// TwinCAT 3 PLC project PLC
// ProgramVersion: 3.1.4026.1+972e9c44872ad038b353624a861fd7e3244e9f75
// libraries:
//   Tc2_Standard, * (Beckhoff Automation GmbH)
//   Tc2_System, * (Beckhoff Automation GmbH)
// project tree:
//   ChainOfResponsibility/ FB_Level1Handler.TcPOU, FB_Level2Handler.TcPOU, FB_Level3Handler.TcPOU, I_Handler.TcIO, PRG_SampleChainOfResponsibility.TcPOU
//   CommandPattern/interfaces/ I_Command.TcIO (not stored)
//   CommandPattern/receiver/ E_ColorCodes.TcDUT
//   CommandPattern/invoker/ FB_RemoteControl.TcPOU
//   CommandPattern/ PRG_SampleCommandPattern.TcPOU
//   CommandPattern/receiver/Light/commands/ FB_CmdLightChangeBrightness.TcPOU, FB_CmdLightChangeColor.TcPOU, FB_CmdLightOff.TcPOU, FB_CmdLightOn.TcPOU
//   CommandPattern/receiver/Light/ FB_Light.TcPOU, I_Light.TcIO
//   Iterator/Collections/ FB_ElementsStation1.TcPOU, FB_ElementsStation2.TcPOU
//   Iterator/Element/ FB_ElementIterator.TcPOU, I_ElementIterator.TcIO, I_IterableElementCollection.TcIO, ST_Element.TcDUT
//   Iterator/ PRG_SampleIterator.TcPOU
//   / MAIN.TcPOU, PlcTask.TcTTO
//   Mediator/Components/Heater/ FB_Heater.TcPOU, I_Heater.TcIO
//   Mediator/Components/SimulateRoomTemperature/ FB_SimulateTemperature.TcPOU
//   Mediator/Components/Thermostat/ FB_Thermostat.TcPOU, I_Thermostat.TcIO
//   Mediator/Mediator/ FB_SmartHome.TcPOU, I_Mediator.TcIO
//   Mediator/ PRG_SampleMediator.TcPOU
//   Memento/Caretaker/ FB_DocumentCaretaker.TcPOU
//   Memento/Memento/ ST_DocumentMemento.TcDUT
//   Memento/Originator/ FB_Document.TcPOU
//   Memento/ PRG_SampleMemento.TcPOU
//   Observer/ PRG_SampleObserver.TcPOU
//   Observer/Publisher/ FB_Publisher.TcPOU
//   Observer/Subscriber/ FB_Subscriber.TcPOU, I_Subscriber.TcIO
//   StatePattern/ FB_StateMachine.TcPOU, PRG_SampleState.TcPOU
//   StatePattern/States/ FB_NotReadyState.TcPOU, FB_ProcessingState.TcPOU, FB_ReadyState.TcPOU, I_State.TcIO
//   Strategy/ FB_TravelTimeCalculator.TcPOU, PRG_SampleStrategy.TcPOU
//   Strategy/Strategies/ FB_StrategyTravelByTrain.TcPOU, FB_StrategyTravelByCar.TcPOU, FB_StrategyTravelByBycicle.TcPOU, I_Strategy.TcIO
//   Visitor/ FB_ElementA.TcPOU, FB_ElementB.TcPOU, FB_Visitor.TcPOU, I_VisitibleElement.TcIO, I_Visitor.TcIO, PRG_SampleVisitor.TcPOU
// real-time tasks:
//   TASK PlcTask: cycle T#10ms, priority 20, ADS port 350

CONFIGURATION PLC
    RESOURCE PLC ON TwinCAT3
        TASK PlcTask(INTERVAL := T#10ms, PRIORITY := 20);
        PROGRAM MAIN WITH PlcTask : MAIN;
    END_RESOURCE
END_CONFIGURATION

// ---- CommandPattern/receiver/E_ColorCodes.TcDUT
{attribute 'qualified_only'}
{attribute 'to_string'}
TYPE E_ColorCodes :
(
	Black 	:= 16#000000,
	Red		:= 16#FF0000,
	Maroon	:= 16#800000,
	Yellow	:= 16#FFFF00,
	Olive	:= 16#808000,
	Lime	:= 16#00FF00,
	Green	:= 16#008000,
	Aqua	:= 16#00FFFF,
	Teal	:= 16#008080,
	Blue	:= 16#0000FF,
	Navy	:= 16#000080,	
	Fuchsia	:= 16#FF00FF,	
	Purple	:= 16#800080,
	White	:= 16#FFFFFF,
	Silver	:= 16#C0C0C0,
	Gray	:= 16#808080
)DWORD;
END_TYPE

// ---- Iterator/Element/ST_Element.TcDUT
TYPE ST_Element :
STRUCT
	sName		:STRING;
END_STRUCT
END_TYPE

// ---- Memento/Memento/ST_DocumentMemento.TcDUT
TYPE ST_DocumentMemento :
STRUCT
	sContent		: STRING;
END_STRUCT
END_TYPE

// ---- ChainOfResponsibility/I_Handler.TcIO
INTERFACE I_Handler

METHOD handleRequest : BOOL
VAR_INPUT
	in_sRequest		: STRING;
END_VAR
END_METHOD

END_INTERFACE

// ---- CommandPattern/receiver/Light/I_Light.TcIO
INTERFACE I_Light

PROPERTY bIsOn : BOOL
GET
END_GET
END_PROPERTY

METHOD changeBrightness : BOOL
VAR_INPUT
	in_rNewBrightness	:REAL;
END_VAR
END_METHOD

METHOD changeColor : BOOL
VAR_INPUT
	in_eNewColor	:E_ColorCodes;
END_VAR
END_METHOD

PROPERTY eColor : E_ColorCodes
GET
END_GET
END_PROPERTY

PROPERTY rBrightness : REAL
GET
END_GET
END_PROPERTY

METHOD turnLightOff : BOOL
VAR_INPUT
END_VAR
END_METHOD

METHOD turnLightOn : BOOL
VAR_INPUT
END_VAR
END_METHOD

END_INTERFACE

// ---- Iterator/Element/I_ElementIterator.TcIO
INTERFACE I_ElementIterator

METHOD hasNext : BOOL
VAR_INPUT
END_VAR
END_METHOD

METHOD init : BOOL
VAR_IN_OUT
	io_astElements	:ARRAY[*] OF ST_Element;
END_VAR
END_METHOD

METHOD next : ST_Element;
VAR_INPUT
END_VAR
END_METHOD

END_INTERFACE

// ---- Iterator/Element/I_IterableElementCollection.TcIO
INTERFACE I_IterableElementCollection

METHOD createIterator : REFERENCE TO FB_ElementIterator
VAR_INPUT
END_VAR
END_METHOD

END_INTERFACE

// ---- Mediator/Components/Heater/I_Heater.TcIO
INTERFACE I_Heater

PROPERTY bIsOn : BOOL
GET
END_GET
END_PROPERTY

PROPERTY sLocation : STRING
GET
END_GET
END_PROPERTY

PROPERTY sName : String
GET
END_GET
END_PROPERTY

METHOD turnOff : Bool
VAR_INPUT
END_VAR
END_METHOD

METHOD turnOn : Bool
VAR_INPUT
END_VAR
END_METHOD

END_INTERFACE

// ---- Mediator/Components/Thermostat/I_Thermostat.TcIO
INTERFACE I_Thermostat

PROPERTY rRequestedTemperature : REAL
GET
END_GET
SET
END_SET
END_PROPERTY

PROPERTY rTemperature : REAL
GET
END_GET
END_PROPERTY

PROPERTY sLocation : STRING
GET
END_GET
END_PROPERTY

PROPERTY sName : String
GET
END_GET
END_PROPERTY

END_INTERFACE

// ---- Mediator/Mediator/I_Mediator.TcIO
INTERFACE I_Mediator

METHOD notify : BOOL
VAR_INPUT
	in_sSenderName		: STRING;
	in_sEvent 			: STRING;
END_VAR
END_METHOD

END_INTERFACE

// ---- Observer/Subscriber/I_Subscriber.TcIO
INTERFACE I_Subscriber

METHOD update : BOOL
VAR_INPUT
	in_sContent			: STRING;
END_VAR
END_METHOD

END_INTERFACE

// ---- StatePattern/States/I_State.TcIO
INTERFACE I_State

PROPERTY CurrentState : STRING
GET
END_GET
END_PROPERTY

METHOD ErrorGone
VAR_INPUT
END_VAR
END_METHOD

METHOD ErrorOccured
VAR_INPUT
END_VAR
END_METHOD

METHOD StartProcess
VAR_INPUT
END_VAR
END_METHOD

METHOD StopProcess
VAR_INPUT
END_VAR
END_METHOD

END_INTERFACE

// ---- Strategy/Strategies/I_Strategy.TcIO
INTERFACE I_Strategy

METHOD execute
VAR_INPUT
	in_rDistance		:REAL;
END_VAR
END_METHOD

END_INTERFACE

// ---- Visitor/I_VisitibleElement.TcIO
INTERFACE I_VisitibleElement

METHOD accept
VAR_INPUT
	in_ipVisitor	: I_Visitor;
END_VAR
END_METHOD

END_INTERFACE

// ---- Visitor/I_Visitor.TcIO
INTERFACE I_Visitor

METHOD VisitElementA
VAR_INPUT
	in_fbElementA		:FB_ElementA;
END_VAR
END_METHOD

METHOD VisitElementB
VAR_INPUT
	in_fbElementB		:FB_ElementB;
END_VAR
END_METHOD

END_INTERFACE

// ---- MAIN.TcPOU
PROGRAM MAIN
VAR
END_VAR

//*************************************************************
// Chain of Responsibility
//*************************************************************
	PRG_SampleChainOfResponsibility();

//*************************************************************
// Command Pattern 
//*************************************************************
	PRG_SampleCommandPattern();
	
//*************************************************************
// Iterator Pattern 
//*************************************************************
	PRG_SampleIterator();

//*************************************************************
// Mediator Pattern 
//*************************************************************
	PRG_SampleMediator();
	
//*************************************************************
// Memento Pattern 
//*************************************************************
	PRG_SampleMemento();
	
//*************************************************************
// Observer Pattern 
//*************************************************************
	PRG_SampleObserver();
	
//*************************************************************
// State Pattern 
//*************************************************************
	PRG_SampleState();	
	
//*************************************************************
// Strategy Pattern 
//*************************************************************
	PRG_SampleStrategy();

END_PROGRAM

// ---- ChainOfResponsibility/PRG_SampleChainOfResponsibility.TcPOU
PROGRAM PRG_SampleChainOfResponsibility
VAR
	fbLvl1Handler			: FB_Level1Handler();
	fbLvl2Handler			: FB_Level2Handler();
	fbLvl3Handler			: FB_Level3Handler();
	
	
	sRequest				: STRING;
	sOldRequest				: STRING;
	bRequestHandled			: BOOL;
	aipHandlers				: ARRAY[0..2] OF I_Handler;
	iCurrentHandlerIndex	: INT;
END_VAR

//*************************************************************
// Call initial Request
//*************************************************************
IF sRequest <> sOldRequest THEN
	sOldRequest := sRequest;
	
	aipHandlers[0] := fbLvl1Handler;
	aipHandlers[1] := fbLvl2Handler;
	aipHandlers[2] := fbLvl3Handler;
	bRequestHandled := FALSE;
	
	FOR iCurrentHandlerIndex:= 0 TO 2 DO
		bRequestHandled := aipHandlers[iCurrentHandlerIndex].handleRequest(in_sRequest := sRequest);
		IF bRequestHandled THEN
			EXIT;
		END_IF
	END_FOR
	
	IF NOT bRequestHandled THEN
		ADSLOGSTR(msgCtrlMask:= ADSLOG_MSGTYPE_ERROR, msgFmtStr:= 'Request cannot be solved by anyone. Request: %s', strArg:= sRequest);
	END_IF
END_IF

END_PROGRAM

// ---- ChainOfResponsibility/FB_Level1Handler.TcPOU
FUNCTION_BLOCK FB_Level1Handler IMPLEMENTS I_Handler
VAR_INPUT
END_VAR
VAR_OUTPUT
END_VAR
VAR
END_VAR

METHOD handleRequest : BOOL
VAR_INPUT
	in_sRequest		: STRING;
END_VAR
handleRequest := FALSE;

IF FIND(in_sRequest, 'Level 1') <> 0 THEN
	ADSLOGSTR(msgCtrlMask:= ADSLOG_MSGTYPE_ERROR, msgFmtStr:= 'Request solved by Level 1. Request: %s', strArg:= in_sRequest);
	handleRequest := TRUE;
ELSE
	ADSLOGSTR(msgCtrlMask:= ADSLOG_MSGTYPE_ERROR, msgFmtStr:= 'Request cannot solved by Level 1. Request: %s', strArg:= in_sRequest);
END_IF
END_METHOD

END_FUNCTION_BLOCK

// ---- ChainOfResponsibility/FB_Level2Handler.TcPOU
FUNCTION_BLOCK FB_Level2Handler IMPLEMENTS I_Handler
VAR_INPUT
END_VAR
VAR_OUTPUT
END_VAR
VAR
END_VAR

METHOD handleRequest : BOOL
VAR_INPUT
	in_sRequest		: STRING;
END_VAR
handleRequest := FALSE;

IF FIND(in_sRequest, 'Level 2') <> 0 THEN
	ADSLOGSTR(msgCtrlMask:= ADSLOG_MSGTYPE_ERROR, msgFmtStr:= 'Request solved by Level 2. Request: %s', strArg:= in_sRequest);
	handleRequest := TRUE;
ELSE
	ADSLOGSTR(msgCtrlMask:= ADSLOG_MSGTYPE_ERROR, msgFmtStr:= 'Request cannot be solved by Level 2. Request: %s', strArg:= in_sRequest);
END_IF
END_METHOD

END_FUNCTION_BLOCK

// ---- ChainOfResponsibility/FB_Level3Handler.TcPOU
FUNCTION_BLOCK FB_Level3Handler IMPLEMENTS I_Handler
VAR_INPUT
END_VAR
VAR_OUTPUT
END_VAR
VAR
END_VAR

METHOD handleRequest : BOOL
VAR_INPUT
	in_sRequest		: STRING;
END_VAR
handleRequest := FALSE;

IF FIND(in_sRequest, 'Level 3') <> 0 THEN
	ADSLOGSTR(msgCtrlMask:= ADSLOG_MSGTYPE_ERROR, msgFmtStr:= 'Request solved by Level 3. Request: %s', strArg:= in_sRequest);
	handleRequest := TRUE;
ELSE
	ADSLOGSTR(msgCtrlMask:= ADSLOG_MSGTYPE_ERROR, msgFmtStr:= 'Request cannot solved by Level 3. Request: %s', strArg:= in_sRequest);
END_IF
END_METHOD

END_FUNCTION_BLOCK

// ---- CommandPattern/PRG_SampleCommandPattern.TcPOU
PROGRAM PRG_SampleCommandPattern
VAR
	fbLight								: FB_Light;
	// Commands
	fbLightOnCmd						: FB_CmdLightOn(ipLight := fbLight);
	fbLightOffCmd						: FB_CmdLightOff(ipLight := fbLight);
	fbIncreaseBrightnessCmd				: FB_CmdLightChangeBrightness(ipLight := fbLight, rBrightnessChange:= 10.0);
	fbDecreaseBrightnessCmd				: FB_CmdLightChangeBrightness(ipLight := fbLight, rBrightnessChange:= -10.0);
	fbChangeColorFav1Cmd				: FB_CmdLightChangeColor(ipLight := fbLight, eColor:= E_ColorCodes.Red);
	fbChangeColorFav2Cmd				: FB_CmdLightChangeColor(ipLight := fbLight, eColor:= E_ColorCodes.Green);
	// Invoker
	fbRemoteControl						: FB_RemoteControl(ipCmdOn:= fbLightOnCmd, ipCmdOff:= fbLightOffCmd, ipCmdFav1:= fbIncreaseBrightnessCmd, ipCmdFav2:= fbDecreaseBrightnessCmd);
	
	// Test events
	bChangeToColorControl				: BOOL;
	bChangeToBrightnessControl			: BOOL;
	
	eOldFav1Color						: E_ColorCodes;
	eFav1Color							: E_ColorCodes;	
	eOldFav2Color						: E_ColorCodes;
	eFav2Color							: E_ColorCodes;
	
	rOldIncreaseSteps					: REAL;
	rIncreaseSteps						: REAL;	
	rOldDecreaseSteps					: REAL;
	rDecreaseSteps						: REAL;	
	
	bPressOn							: BOOL;
	bPressOff							: BOOL;
	bPressFav1							: BOOL;
	bPressFav2							: BOOL;
END_VAR

//*************************************************************
// Call Object Light
//*************************************************************
	fbLight();

//*************************************************************
// Change Functionality of Remote Control
//*************************************************************

	//*************************************************************
	// Color control
	//*************************************************************
	IF bChangeToColorControl THEN
		bChangeToColorControl := FALSE;
		fbRemoteControl.setCommands(
										in_ipCmdOn		:= fbLightOnCmd, 
										in_ipCmdOff		:= fbLightOffCmd, 
										in_ipCmdFav1	:= fbChangeColorFav1Cmd, 
										in_ipCmdFav2	:= fbChangeColorFav2Cmd);
	END_IF
	
	IF eFav1Color <> eOldFav1Color THEN
		eOldFav1Color := eFav1Color;
		fbChangeColorFav1Cmd.setChangeColor(in_eNewChangeColor := eFav1Color);
	END_IF
	
	IF eFav2Color <> eOldFav2Color THEN
		eOldFav2Color := eFav2Color;
		fbChangeColorFav2Cmd.setChangeColor(in_eNewChangeColor := eFav2Color);
	END_IF
	
	//*************************************************************
	// Brightness control
	//*************************************************************
	IF bChangeToBrightnessControl THEN
		bChangeToBrightnessControl := FALSE;
		fbRemoteControl.setCommands(
										in_ipCmdOn		:= fbLightOnCmd, 
										in_ipCmdOff		:= fbLightOffCmd, 
										in_ipCmdFav1	:= fbIncreaseBrightnessCmd, 
										in_ipCmdFav2	:= fbDecreaseBrightnessCmd);
	END_IF
	
	IF rIncreaseSteps <> rOldIncreaseSteps THEN
		rOldIncreaseSteps := rIncreaseSteps;
		fbIncreaseBrightnessCmd.setChangeBrightness(in_rNewChangeBrightness := rIncreaseSteps);
	END_IF
	
	IF rDecreaseSteps <> rOldDecreaseSteps THEN
		rOldDecreaseSteps := rDecreaseSteps;
		fbDecreaseBrightnessCmd.setChangeBrightness(in_rNewChangeBrightness := rDecreaseSteps);
	END_IF

//*************************************************************
// Do Actions
//*************************************************************
	IF bPressOn THEN
		bPressOn := FALSE;
		fbRemoteControl.pressOn();
	END_IF
	
	IF bPressOff THEN
		bPressOff := FALSE;
		fbRemoteControl.pressOff();
	END_IF
	
	IF bPressFav1 THEN
		bPressFav1 := FALSE;
		fbRemoteControl.pressFav1();
	END_IF
	
	IF bPressFav2 THEN
		bPressFav2 := FALSE;
		fbRemoteControl.pressFav2();
	END_IF

END_PROGRAM

// ---- CommandPattern/receiver/Light/FB_Light.TcPOU
FUNCTION_BLOCK FB_Light IMPLEMENTS I_LIGHT
VAR_INPUT
END_VAR
VAR_OUTPUT
END_VAR
VAR
	_rBrightness	: REAL;
	_eColor			: E_ColorCodes;
	_bIsOn			: BOOL;
END_VAR

PROPERTY bIsOn : BOOL
GET
bIsOn := _bIsOn;
END_GET
END_PROPERTY

METHOD changeBrightness : BOOL
VAR_INPUT
	in_rNewBrightness	: REAL;
END_VAR
IF in_rNewBrightness > 100.0 THEN
	_rBrightness := 100.0;
ELSIF in_rNewBrightness < 0.0 THEN
	_rBrightness := 0.0;
ELSE
	_rBrightness := in_rNewBrightness;
END_IF

ADSLOGSTR(msgCtrlMask:= ADSLOG_MSGTYPE_ERROR, msgFmtStr:= 'New Brightness: %s', strArg:= TO_STRING(_rBrightness));
END_METHOD

METHOD changeColor : BOOL
VAR_INPUT
	in_eNewColor	:E_ColorCodes;
END_VAR
_eColor := in_eNewColor;
ADSLOGSTR(msgCtrlMask:= ADSLOG_MSGTYPE_ERROR, msgFmtStr:= 'New Color: %s', strArg:= TO_STRING(_eColor));
END_METHOD

PROPERTY eColor : E_ColorCodes
GET
eColor := _eColor;
END_GET
END_PROPERTY

PROPERTY rBrightness : REAL
GET
rBrightness := _rBrightness;
END_GET
END_PROPERTY

METHOD turnLightOff : BOOL
VAR_INPUT
END_VAR
_bIsOn := FALSE;
ADSLOGSTR(msgCtrlMask:= ADSLOG_MSGTYPE_ERROR, msgFmtStr:= 'Light is off', strArg:= '');
ADSLOGSTR(msgCtrlMask:= ADSLOG_MSGTYPE_ERROR, msgFmtStr:= 'Brightness: %s', strArg:= TO_STRING(_rBrightness));
ADSLOGSTR(msgCtrlMask:= ADSLOG_MSGTYPE_ERROR, msgFmtStr:= 'Color: %s', strArg:= TO_STRING(_eColor));
END_METHOD

METHOD turnLightOn : BOOL
VAR_INPUT
END_VAR
_bIsOn := TRUE;

IF _rBrightness <= 0.0 THEN
	_rBrightness := 100.0;
END_IF

IF _eColor = E_ColorCodes.Black THEN
	_eColor := E_ColorCodes.White;
END_IF

ADSLOGSTR(msgCtrlMask:= ADSLOG_MSGTYPE_ERROR, msgFmtStr:= 'Light is on', strArg:= '');
ADSLOGSTR(msgCtrlMask:= ADSLOG_MSGTYPE_ERROR, msgFmtStr:= 'Brightness: %s', strArg:= TO_STRING(_rBrightness));
ADSLOGSTR(msgCtrlMask:= ADSLOG_MSGTYPE_ERROR, msgFmtStr:= 'Color: %s', strArg:= TO_STRING(_eColor));
END_METHOD

END_FUNCTION_BLOCK

// ---- CommandPattern/receiver/Light/commands/FB_CmdLightOn.TcPOU
FUNCTION_BLOCK FB_CmdLightOn IMPLEMENTS I_Command
VAR_INPUT
END_VAR
VAR_OUTPUT
END_VAR
VAR
	_ipLight				: I_Light;
END_VAR

METHOD execute : BOOL
_ipLight.turnLightOn();
END_METHOD

//FB_Init is always available implicitly and it is used primarily for initialization.
//The return value is not evaluated. For a specific influence, you can also declare the
//methods explicitly and provide additional code there with the standard initialization
//code. You can evaluate the return value.
METHOD FB_Init: BOOL
VAR_INPUT
    bInitRetains: BOOL; // TRUE: the retain variables are initialized (reset warm / reset cold)
    bInCopyCode: BOOL;  // TRUE: the instance will be copied to the copy code afterward (online change)   
	ipLight: I_Light;
END_VAR
_ipLight := ipLight;
END_METHOD

END_FUNCTION_BLOCK

// ---- CommandPattern/receiver/Light/commands/FB_CmdLightOff.TcPOU
FUNCTION_BLOCK FB_CmdLightOff IMPLEMENTS I_Command
VAR_INPUT
END_VAR
VAR_OUTPUT
END_VAR
VAR
	_ipLight				: I_Light;
END_VAR

METHOD execute : BOOL
_ipLight.turnLightOff();
END_METHOD

//FB_Init is always available implicitly and it is used primarily for initialization.
//The return value is not evaluated. For a specific influence, you can also declare the
//methods explicitly and provide additional code there with the standard initialization
//code. You can evaluate the return value.
METHOD FB_Init: BOOL
VAR_INPUT
    bInitRetains: BOOL; // TRUE: the retain variables are initialized (reset warm / reset cold)
    bInCopyCode: BOOL;  // TRUE: the instance will be copied to the copy code afterward (online change)   
	ipLight: I_Light;
END_VAR
_ipLight := ipLight;
END_METHOD

END_FUNCTION_BLOCK

// ---- CommandPattern/receiver/Light/commands/FB_CmdLightChangeBrightness.TcPOU
FUNCTION_BLOCK FB_CmdLightChangeBrightness IMPLEMENTS I_Command
VAR_INPUT
END_VAR
VAR_OUTPUT
END_VAR
VAR
	_rBrightnessChange		: REAL;
	_ipLight				: I_Light;
END_VAR

METHOD execute : BOOL
_ipLight.changeBrightness(in_rNewBrightness:= (_ipLight.rBrightness + _rBrightnessChange));
END_METHOD

//FB_Init is always available implicitly and it is used primarily for initialization.
//The return value is not evaluated. For a specific influence, you can also declare the
//methods explicitly and provide additional code there with the standard initialization
//code. You can evaluate the return value.
METHOD FB_Init: BOOL
VAR_INPUT
    bInitRetains: BOOL; // TRUE: the retain variables are initialized (reset warm / reset cold)
    bInCopyCode: BOOL;  // TRUE: the instance will be copied to the copy code afterward (online change)   
	rBrightnessChange :REAL;
	ipLight: I_Light;
END_VAR
_ipLight := ipLight;
_rBrightnessChange := rBrightnessChange;
END_METHOD

METHOD setChangeBrightness : BOOL
VAR_INPUT
	in_rNewChangeBrightness	: REAL;
END_VAR
_rBrightnessChange := in_rNewChangeBrightness;
END_METHOD

END_FUNCTION_BLOCK

// ---- CommandPattern/receiver/Light/commands/FB_CmdLightChangeColor.TcPOU
FUNCTION_BLOCK FB_CmdLightChangeColor IMPLEMENTS I_Command
VAR_INPUT
END_VAR
VAR_OUTPUT
END_VAR
VAR
	_eChangeColor			: E_ColorCodes;
	_ipLight				: I_Light;
END_VAR

METHOD execute : BOOL
_ipLight.changeColor(in_eNewColor:= _eChangeColor);
END_METHOD

//FB_Init is always available implicitly and it is used primarily for initialization.
//The return value is not evaluated. For a specific influence, you can also declare the
//methods explicitly and provide additional code there with the standard initialization
//code. You can evaluate the return value.
METHOD FB_Init: BOOL
VAR_INPUT
    bInitRetains: BOOL; // TRUE: the retain variables are initialized (reset warm / reset cold)
    bInCopyCode: BOOL;  // TRUE: the instance will be copied to the copy code afterward (online change)   
	eColor : E_ColorCodes;
	ipLight: I_Light;
END_VAR
_ipLight := ipLight;
_eChangeColor := eColor;
END_METHOD

METHOD setChangeColor : BOOL
VAR_INPUT
	in_eNewChangeColor	: E_ColorCodes;
END_VAR
_eChangeColor := in_eNewChangeColor;
END_METHOD

END_FUNCTION_BLOCK

// ---- CommandPattern/invoker/FB_RemoteControl.TcPOU
FUNCTION_BLOCK FB_RemoteControl
VAR_INPUT
END_VAR
VAR_OUTPUT
END_VAR
VAR
	_ipCmdOn		: I_Command;
	_ipCmdOff		: I_Command;
	_ipCmdFav1		: I_Command;
	_ipCmdFav2		: I_Command;
END_VAR

//FB_Init is always available implicitly and it is used primarily for initialization.
//The return value is not evaluated. For a specific influence, you can also declare the
//methods explicitly and provide additional code there with the standard initialization
//code. You can evaluate the return value.
METHOD FB_Init: BOOL
VAR_INPUT
    bInitRetains: BOOL; // TRUE: the retain variables are initialized (reset warm / reset cold)
    bInCopyCode: BOOL;  // TRUE: the instance will be copied to the copy code afterward (online change)   
	ipCmdOn		: I_Command;
	ipCmdOff	: I_Command;
	ipCmdFav1	: I_Command;
	ipCmdFav2	: I_Command;
END_VAR
_ipCmdOn		:= ipCmdOn;
_ipCmdOff		:= ipCmdOff;
_ipCmdFav1		:= ipCmdFav1;
_ipCmdFav2		:= ipCmdFav2;
END_METHOD

METHOD pressFav1 : BOOL
VAR_INPUT
END_VAR
_ipCmdFav1.execute();
END_METHOD

METHOD pressFav2 : BOOL
VAR_INPUT
END_VAR
_ipCmdFav2.execute();
END_METHOD

METHOD pressOff : BOOL
VAR_INPUT
END_VAR
_ipCmdOff.execute();
END_METHOD

METHOD pressOn : BOOL
VAR_INPUT
END_VAR
_ipCmdOn.execute();
END_METHOD

METHOD setCommands : BOOL
VAR_INPUT
	in_ipCmdOn		: I_Command;
	in_ipCmdOff		: I_Command;
	in_ipCmdFav1	: I_Command;
	in_ipCmdFav2	: I_Command;
END_VAR
_ipCmdOn		:= in_ipCmdOn;
_ipCmdOff		:= in_ipCmdOff;
_ipCmdFav1		:= in_ipCmdFav1;
_ipCmdFav2		:= in_ipCmdFav2;
END_METHOD

END_FUNCTION_BLOCK

// ---- Iterator/PRG_SampleIterator.TcPOU
PROGRAM PRG_SampleIterator
VAR
	fbElementsStation1				: FB_ElementsStation1;
	fbElementStation1Iterator   	: REFERENCE TO FB_ElementIterator;
	fbElementsStation2				: FB_ElementsStation2;
	fbElementStation2Iterator   	: REFERENCE TO FB_ElementIterator;
	
	bIterateStation1				: BOOL;
	bIterateStation2				: BOOL;
END_VAR

VAR_TEMP
	stElement						:ST_Element;
END_VAR

fbElementsStation1();
fbElementsStation2();


IF bIterateStation1 THEN
	bIterateStation1 := FALSE;
	
	fbElementStation1Iterator REF= fbElementsStation1.createIterator();
	WHILE fbElementStation1Iterator.hasNext() DO
		stElement := fbElementStation1Iterator.next();
		ADSLOGSTR(msgCtrlMask:= ADSLOG_MSGTYPE_ERROR, msgFmtStr:= '%s found.', strArg:= stElement.sName);
	END_WHILE
END_IF

IF bIterateStation2 THEN
	bIterateStation2 := FALSE;
	
	fbElementStation2Iterator REF= fbElementsStation2.createIterator();
	WHILE fbElementStation2Iterator.hasNext() DO
		stElement := fbElementStation2Iterator.next();
		ADSLOGSTR(msgCtrlMask:= ADSLOG_MSGTYPE_ERROR, msgFmtStr:= '%s found.', strArg:= stElement.sName);
	END_WHILE
END_IF

END_PROGRAM

// ---- Iterator/Collections/FB_ElementsStation1.TcPOU
FUNCTION_BLOCK FB_ElementsStation1 IMPLEMENTS I_IterableElementCollection
VAR_INPUT
END_VAR
VAR_OUTPUT
END_VAR
VAR
	_astElements			: ARRAY[0..MAX_ELEMENTS] OF ST_Element;	
	_fbIterator				: FB_ElementIterator;
END_VAR

VAR CONSTANT
	MAX_ELEMENTS			: INT := 30;
END_VAR

METHOD createIterator : REFERENCE TO FB_ElementIterator
_fbIterator.init(io_astElements := _astElements);
createIterator REF= _fbIterator;
END_METHOD

//FB_Init is always available implicitly and it is used primarily for initialization.
//The return value is not evaluated. For a specific influence, you can also declare the
//methods explicitly and provide additional code there with the standard initialization
//code. You can evaluate the return value.
METHOD FB_Init: BOOL
VAR_INPUT
    bInitRetains: BOOL; // TRUE: the retain variables are initialized (reset warm / reset cold)
    bInCopyCode: BOOL;  // TRUE: the instance will be copied to the copy code afterward (online change)   
END_VAR
VAR 
	i : INT;
END_VAR
FOR i:= 0 TO MAX_ELEMENTS DO
	_astElements[i].sName:= CONCAT('Element Station 1 No: ', TO_STRING(i + 1));
END_FOR
END_METHOD

END_FUNCTION_BLOCK

// ---- Iterator/Element/FB_ElementIterator.TcPOU
FUNCTION_BLOCK FB_ElementIterator IMPLEMENTS I_ElementIterator
VAR_INPUT
END_VAR
VAR_OUTPUT
END_VAR
VAR
	_pElementData		: POINTER TO ST_Element;
	_diNumOfElements	: DINT;
	_diIndex			: DINT;
END_VAR

METHOD hasNext : BOOL
VAR
	
END_VAR
IF _pElementData = 0 THEN
	RETURN;
END_IF

hasNext := _diIndex < _diNumOfElements;
END_METHOD

METHOD init : BOOL
VAR_IN_OUT
	io_astElements	:ARRAY[*] OF ST_Element;
END_VAR
_pElementData 		:= io_astElements;
_diNumOfElements 	:= UPPER_BOUND(io_astElements, 1);
_diIndex			:= LOWER_BOUND(io_astElements, 1);
END_METHOD

METHOD next : ST_Element
VAR
	stElement :ST_Element;
END_VAR
IF _pElementData = 0 THEN
	RETURN;
END_IF

IF _diIndex < _diNumOfElements THEN
	MEMCPY(srcAddr:= (_pElementData + (_diIndex * SIZEOF(stElement))), destAddr:= ADR(stElement), n:= SIZEOF(stElement));
	next := stElement;
	_diIndex := _diIndex + 1;
END_IF
END_METHOD

END_FUNCTION_BLOCK

// ---- Iterator/Collections/FB_ElementsStation2.TcPOU
FUNCTION_BLOCK FB_ElementsStation2 IMPLEMENTS I_IterableElementCollection
VAR_INPUT
END_VAR
VAR_OUTPUT
END_VAR
VAR
	_astElements			: ARRAY[0..MAX_ELEMENTS] OF ST_Element;
	_fbIterator				: FB_ElementIterator;
END_VAR

VAR CONSTANT
	MAX_ELEMENTS			: INT := 5;
END_VAR

METHOD createIterator : REFERENCE TO FB_ElementIterator
_fbIterator.init(io_astElements := _astElements);
createIterator REF= _fbIterator;
END_METHOD

//FB_Init is always available implicitly and it is used primarily for initialization.
//The return value is not evaluated. For a specific influence, you can also declare the
//methods explicitly and provide additional code there with the standard initialization
//code. You can evaluate the return value.
METHOD FB_Init: BOOL
VAR_INPUT
    bInitRetains: BOOL; // TRUE: the retain variables are initialized (reset warm / reset cold)
    bInCopyCode: BOOL;  // TRUE: the instance will be copied to the copy code afterward (online change)   
END_VAR
VAR 
	i : INT;
END_VAR
FOR i:= 0 TO MAX_ELEMENTS DO
	_astElements[i].sName:= CONCAT('Element Station 2 No: ', TO_STRING(i + 1));
END_FOR
END_METHOD

END_FUNCTION_BLOCK

// ---- Mediator/PRG_SampleMediator.TcPOU
PROGRAM PRG_SampleMediator
VAR
	fbSmartHomeDevice			:FB_SmartHome;	

	fbHeaterKitchen				:FB_Heater(sName:= 'Heater', sLocation := 'Kitchen', ipMediator:= fbSmartHomeDevice);
	fbHeaterBedroom				:FB_Heater(sName:= 'Heater', sLocation := 'Bedroom', ipMediator:= fbSmartHomeDevice);
	
	fbThermostatKitchen			:FB_Thermostat(sName:= 'Thermostat', sLocation := 'Kitchen', rRequestedTemperature := 20.0, ipMediator:= fbSmartHomeDevice);
	fbThermostatBedroom			:FB_Thermostat(sName:= 'Door', sLocation := 'Bedroom', rRequestedTemperature := 14.0, ipMediator:= fbSmartHomeDevice);
	
	fbRoomTempKitchen			:FB_SimulateTemperature;
	fbRoomTempBedroom			:FB_SimulateTemperature;
	
	bEnable						:BOOL;
	bAddAllDevices				:BOOL := TRUE; // Event to add all devices to Mediator
	bRemoveAllDevices			:BOOL;
END_VAR

//*************************************************************
// Disable Test enviroment
//*************************************************************	
	IF NOT bEnable THEN
		
		RETURN;
		
	END_IF

//*************************************************************
// Call Objects
//*************************************************************
	fbSmartHomeDevice();
	
	fbHeaterKitchen();
	fbHeaterBedroom();
	
	fbThermostatKitchen(in_rTemperature := fbRoomTempKitchen.out_bSimTemperature);
	fbThermostatBedroom(in_rTemperature := fbRoomTempBedroom.out_bSimTemperature);
	
	fbRoomTempKitchen(in_bTempShouldRise := fbHeaterKitchen.bIsOn);
	fbRoomTempBedroom(in_bTempShouldRise := fbHeaterBedroom.bIsOn);
	
//*************************************************************
// Add Objects to Smart Home Device
//*************************************************************	
IF bAddAllDevices THEN
	
	bAddAllDevices := FALSE;
	
	fbSmartHomeDevice.addHeater(fbHeaterKitchen);
	//fbSmartHomeDevice.addHeater(fbHeaterBedroom);
	
	fbSmartHomeDevice.addThermostat(fbThermostatKitchen);
	//fbSmartHomeDevice.addThermostat(fbThermostatBedroom);
	
END_IF

IF bRemoveAllDevices THEN
	
	bRemoveAllDevices := FALSE;
	
	fbSmartHomeDevice.removeHeater(fbHeaterKitchen);
	fbSmartHomeDevice.removeHeater(fbHeaterBedroom);
	
	fbSmartHomeDevice.removeThermostat(fbThermostatKitchen);
	fbSmartHomeDevice.removeThermostat(fbThermostatBedroom);
	
END_IF

END_PROGRAM

// ---- Mediator/Mediator/FB_SmartHome.TcPOU
FUNCTION_BLOCK FB_SmartHome IMPLEMENTS I_Mediator
VAR_INPUT
END_VAR
VAR_OUTPUT
END_VAR
VAR
	_aipHeater				: ARRAY [0..MAX_HEATER] OF I_Heater;
	_aipThermostat			: ARRAY [0..MAX_THERMOSTAT] OF I_Thermostat;
END_VAR
VAR CONSTANT
	MAX_HEATER				: INT := 5;
	MAX_THERMOSTAT			: INT := 10;
END_VAR

METHOD addHeater : BOOL
VAR_INPUT
	in_ipHeater		: I_Heater;
END_VAR

VAR
	bAdded	: BOOL;
	i		: INT;
END_VAR
addHeater := FALSE;

FOR i := 0 TO (MAX_HEATER - 1) DO
	
	IF _aipHeater[i] = 0 THEN
		
		_aipHeater[i] := in_ipHeater;
		addHeater := TRUE;
		EXIT;
		
	END_IF
	
END_FOR
END_METHOD

METHOD addThermostat : BOOL
VAR_INPUT
	in_ipThermostat		: I_Thermostat;
END_VAR

VAR
	i		: INT;
END_VAR
addThermostat := FALSE;

FOR i := 0 TO (MAX_THERMOSTAT - 1) DO
	
	IF _aipThermostat[i] = 0 THEN
		
		_aipThermostat[i] := in_ipThermostat;
		addThermostat := TRUE;
		EXIT;
		
	END_IF
	
END_FOR
END_METHOD

METHOD PRIVATE getHeaterByLocation : BOOL
VAR_INPUT
	in_sLocation 		: STRING;
END_VAR
VAR_OUTPUT
	out_ipHeater		: I_Heater;
END_VAR

VAR
	i					: INT;
END_VAR
// Init
getHeaterByLocation 	:= FALSE;
out_ipHeater		:= 0;

// Loop through list
FOR i:= 0 TO (MAX_HEATER - 1) DO
	
	// Check if interface is valid
	IF _aipHeater[i] = 0 THEN
		
		CONTINUE;
		
	END_IF
	
	IF _aipHeater[i].sLocation = in_sLocation THEN
		
		getHeaterByLocation := TRUE;
		out_ipHeater := _aipHeater[i];
		RETURN;
		
	END_IF
	
END_FOR
END_METHOD

METHOD PRIVATE getHeaterByName : BOOL
VAR_INPUT
	in_sSenderName 		: STRING;
END_VAR
VAR_OUTPUT
	out_ipHeater		: I_Heater;
END_VAR

VAR
	i					: INT;
END_VAR
// Init
getHeaterByName 	:= FALSE;
out_ipHeater		:= 0;

// Loop through list
FOR i:= 0 TO (MAX_HEATER - 1) DO
	
	// Check if interface is valid
	IF _aipHeater[i] = 0 THEN
		
		CONTINUE;
		
	END_IF
	
	IF _aipHeater[i].sName = in_sSenderName THEN
		
		getHeaterByName := TRUE;
		out_ipHeater := _aipHeater[i];
		RETURN;
		
	END_IF
	
END_FOR
END_METHOD

METHOD PRIVATE getThermostatByName : BOOL
VAR_INPUT
	in_sSenderName 		: STRING;
END_VAR
VAR_OUTPUT
	out_ipThermostat	: I_Thermostat;
END_VAR

VAR
	i					: INT;
END_VAR
// Init
getThermostatByName 	:= FALSE;
out_ipThermostat	:= 0;

// Loop through list
FOR i:= 0 TO (MAX_THERMOSTAT - 1) DO
	
	// Check if interface is valid
	IF _aipThermostat[i] = 0 THEN
		
		CONTINUE;
		
	END_IF
	
	IF _aipThermostat[i].sName = in_sSenderName THEN
		
		getThermostatByName := TRUE;
		out_ipThermostat := _aipThermostat[i];
		RETURN;
		
	END_IF
	
END_FOR
END_METHOD

METHOD notify : BOOL
VAR_INPUT
	in_sSenderName		: STRING;
	in_sEvent			: STRING;
END_VAR

VAR
	i					: INT;
	ipTmpThermostat		: I_Thermostat;
	ipTmpHeater			: I_Heater;
END_VAR
//*************************************************************
// This is the point where the logic happens
//*************************************************************

// Check if sender is Heater
IF getHeaterByName(in_sSenderName := in_sSenderName, out_ipHeater => ipTmpHeater) THEN
	
	// nothing to do here
	RETURN;
	
END_IF

// Check if sender is Thermostat
IF getThermostatByName(in_sSenderName := in_sSenderName, out_ipThermostat => ipTmpThermostat) THEN
	
	// Check evenet
	IF in_sEvent = 'It is to cold' THEN	
		
		// Decide which heater needs to be turned on		
		IF getHeaterByLocation(in_sLocation := ipTmpThermostat.sLocation, out_ipHeater => ipTmpHeater) THEN
			
			ipTmpHeater.turnOn();
			
		END_IF
		
	ELSIF in_sEvent = 'It is to warm' THEN
		
		// Decide which heater needs to be turned on		
		IF getHeaterByLocation(in_sLocation := ipTmpThermostat.sLocation, out_ipHeater => ipTmpHeater) THEN
			
			ipTmpHeater.turnOff();
			
		END_IF
		
	END_IF
END_IF
END_METHOD

METHOD removeHeater : BOOL
VAR_INPUT
	in_ipHeater		: I_Heater;
END_VAR

VAR
	i		: INT;
END_VAR
removeHeater := FALSE;

FOR i := 0 TO (MAX_HEATER - 1) DO
	
	IF _aipHeater[i] = in_ipHeater THEN
		
		_aipHeater[i] := 0;
		removeHeater := TRUE;
		EXIT;
		
	END_IF
	
END_FOR
END_METHOD

METHOD removeThermostat : BOOL
VAR_INPUT
	in_ipThermostat		: I_Thermostat;
END_VAR

VAR
	i		: INT;
END_VAR
removeThermostat := FALSE;

FOR i := 0 TO (MAX_THERMOSTAT - 1) DO
	
	IF _aipThermostat[i] = in_ipThermostat THEN
		
		_aipThermostat[i] := 0;
		removeThermostat := TRUE;
		EXIT;
		
	END_IF
	
END_FOR
END_METHOD

END_FUNCTION_BLOCK

// ---- Mediator/Components/Heater/FB_Heater.TcPOU
FUNCTION_BLOCK FB_Heater IMPLEMENTS I_Heater
VAR_INPUT
END_VAR
VAR_OUTPUT	
END_VAR
VAR
	_sName				: STRING;
	_sLocation			: STRING;
	_bIsOn				: BOOL;
	_ipMediator			: I_Mediator;
END_VAR

PROPERTY bIsOn : Bool
GET
bIsOn := _bIsOn;
END_GET
END_PROPERTY

//FB_Init is always available implicitly and it is used primarily for initialization.
//The return value is not evaluated. For a specific influence, you can also declare the
//methods explicitly and provide additional code there with the standard initialization
//code. You can evaluate the return value.
METHOD FB_Init: BOOL
VAR_INPUT
    bInitRetains: BOOL; // TRUE: the retain variables are initialized (reset warm / reset cold)
    bInCopyCode: BOOL;  // TRUE: the instance will be copied to the copy code afterward (online change)  
	sName: STRING;
	sLocation: STRING;
	ipMediator: I_Mediator; 
END_VAR
_ipMediator := ipMediator;
_sName := sName;
_sLocation := sLocation;
END_METHOD

{warning 'Add property implementation'}
PROPERTY sLocation : STRING
GET
sLocation := _sLocation;
END_GET
END_PROPERTY

{warning 'Add property implementation'}
PROPERTY sName : STRING
GET
sName := _sName;
END_GET
END_PROPERTY

METHOD turnOff : BOOL
VAR_INPUT
END_VAR
IF NOT _bIsOn THEN
	
	RETURN;

END_IF


_bIsOn := FALSE;
ADSLOGSTR(msgCtrlMask:= ADSLOG_MSGTYPE_ERROR, msgFmtStr:= '%s turned heater off.', strArg:= CONCAT(_sName, CONCAT('|', _sLocation)));

// Notify moderator about the event
_ipMediator.notify(in_sSenderName:= _sName, in_sEvent := 'Heater off');
END_METHOD

METHOD turnOn : BOOL
VAR_INPUT
END_VAR
IF _bIsOn THEN
	
	RETURN;

END_IF

_bIsOn := TRUE;
ADSLOGSTR(msgCtrlMask:= ADSLOG_MSGTYPE_ERROR, msgFmtStr:= '%s turned heater on.', strArg:= CONCAT(_sName, CONCAT('|', _sLocation)));

// Notify moderator about the event
_ipMediator.notify(in_sSenderName:= _sName, in_sEvent := 'Heater on');
END_METHOD

END_FUNCTION_BLOCK

// ---- Mediator/Components/Thermostat/FB_Thermostat.TcPOU
FUNCTION_BLOCK FB_Thermostat IMPLEMENTS I_Thermostat
VAR_INPUT
	in_rTemperature		: REAL;
END_VAR
VAR_OUTPUT
END_VAR
VAR
	_sName					: STRING;
	_sLocation				: STRING;
	_rTemperature			: REAL;
	_rRequestedTemperature  : REAL;
	_ipMediator				: I_Mediator;
	_fbSamplingRate			: TON;
END_VAR

// Sampling Rate
_fbSamplingRate(IN:= NOT _fbSamplingRate.Q, PT := T#2S);

IF NOT _fbSamplingRate.Q THEN
	RETURN;
END_IF

// Check Temperature changed
IF in_rTemperature <> _rTemperature THEN
	
	_rTemperature := in_rTemperature;	
	_ipMediator.notify(in_sSenderName:= _sName, in_sEvent := 'Temperature changed');
	ADSLOGSTR(msgCtrlMask:= ADSLOG_MSGTYPE_ERROR, msgFmtStr:= '%s temperature changed.', strArg:= CONCAT(_sName, CONCAT(' | ', CONCAT(_sLocation, CONCAT(' | ', TO_STRING(_rTemperature))))));
	
END_IF

// Check Temperature dropped
IF _rTemperature < _rRequestedTemperature THEN
	
	_ipMediator.notify(in_sSenderName:= _sName, in_sEvent := 'It is to cold');
	
END_IF

// Check Temperature rised
IF _rTemperature > _rRequestedTemperature THEN
	
	_ipMediator.notify(in_sSenderName:= _sName, in_sEvent := 'It is to warm');
	
END_IF

//FB_Init is always available implicitly and it is used primarily for initialization.
//The return value is not evaluated. For a specific influence, you can also declare the
//methods explicitly and provide additional code there with the standard initialization
//code. You can evaluate the return value.
METHOD FB_Init: BOOL
VAR_INPUT
    bInitRetains: BOOL; // TRUE: the retain variables are initialized (reset warm / reset cold)
    bInCopyCode: BOOL;  // TRUE: the instance will be copied to the copy code afterward (online change)  
	sName: STRING;
	sLocation: STRING;
	rRequestedTemperature : REAL;
	ipMediator: I_Mediator; 
END_VAR
_ipMediator := ipMediator;
_sName := sName;
_sLocation := sLocation;
_rRequestedTemperature := rRequestedTemperature;
END_METHOD

{warning 'Add property implementation'}
PROPERTY rRequestedTemperature : REAL
GET
END_GET
SET
END_SET
END_PROPERTY

PROPERTY rTemperature : REAL
GET
rTemperature := _rTemperature;
END_GET
END_PROPERTY

{warning 'Add property implementation'}
PROPERTY sLocation : STRING
GET
sLocation := _sLocation;
END_GET
END_PROPERTY

{warning 'Add property implementation'}
PROPERTY sName : STRING
GET
sName := _sName;
END_GET
END_PROPERTY

END_FUNCTION_BLOCK

// ---- Mediator/Components/SimulateRoomTemperature/FB_SimulateTemperature.TcPOU
FUNCTION_BLOCK FB_SimulateTemperature
VAR_INPUT
	in_bTempShouldRise	: BOOL;
END_VAR
VAR_OUTPUT
	out_bSimTemperature	: REAL;
END_VAR
VAR
	_fbChangingRate			: TON;
END_VAR

// Changing Rate
_fbChangingRate(IN:= NOT _fbChangingRate.Q, PT := T#1S);

IF NOT _fbChangingRate.Q THEN
	RETURN;
END_IF

IF in_bTempShouldRise THEN
	
	IF out_bSimTemperature < 30.0 THEN
		
		out_bSimTemperature := out_bSimTemperature + 1;

	END_IF	
	
ELSE

	IF out_bSimTemperature > 8.0 THEN
		
		out_bSimTemperature := out_bSimTemperature - 1;

	END_IF	

END_IF

END_FUNCTION_BLOCK

// ---- Memento/PRG_SampleMemento.TcPOU
PROGRAM PRG_SampleMemento
VAR
	fbDocument			: FB_Document;
	fbHistory			: FB_DocumentCaretaker;
	
	sNewText			: STRING;
	sOldText			: STRING;
	sActText			: STRING;
	
	bUndo				: BOOL;
	bRedo				: BOOL;
END_VAR

//*************************************************************
// Add a new Text to the Document
//*************************************************************	
sActText := fbDocument.sContent; // Actual Text just for debugging

IF sNewText <> sOldText THEN
	
	sOldText := sNewText;
	fbDocument.write(sNewText);
	fbHistory.addMemento(fbDocument.takeSnapshot());
	
END_IF

//*************************************************************
// Undo/ Redo actions
//*************************************************************	
IF bUndo THEN
	
	bUndo := FALSE;
	fbDocument.restoreFromMemento(fbHistory.undoMemento());
	
END_IF

IF bRedo THEN
	
	bRedo := FALSE;
	fbDocument.restoreFromMemento(fbHistory.redoMemento());
	
END_IF

END_PROGRAM

// ---- Memento/Originator/FB_Document.TcPOU
FUNCTION_BLOCK FB_Document
VAR_INPUT
END_VAR
VAR_OUTPUT
END_VAR
VAR
	_sContent		:STRING;
END_VAR

METHOD restoreFromMemento : BOOL
VAR_INPUT
	in_rstMemento		: REFERENCE TO ST_DocumentMemento;
END_VAR
IF NOT __ISVALIDREF(in_rstMemento) THEN
	RETURN;
END_IF

_sContent := in_rstMemento.sContent;

ADSLOGSTR(msgCtrlMask:= ADSLOG_MSGTYPE_ERROR, msgFmtStr:= 'Memento restored. Content: %s', strArg:= _sContent);
END_METHOD

PROPERTY sContent : String
GET
sContent := _sContent;
END_GET
END_PROPERTY

METHOD takeSnapshot : ST_DocumentMemento
takeSnapshot.sContent := _sContent;

ADSLOGSTR(msgCtrlMask:= ADSLOG_MSGTYPE_ERROR, msgFmtStr:= 'New Memento created. Content: %s', strArg:= _sContent);
END_METHOD

METHOD write : BOOL
VAR_INPUT
	in_sText	: STRING;
END_VAR
_sContent := in_sText;
END_METHOD

END_FUNCTION_BLOCK

// ---- Memento/Caretaker/FB_DocumentCaretaker.TcPOU
FUNCTION_BLOCK FB_DocumentCaretaker
VAR_INPUT
END_VAR
VAR_OUTPUT
END_VAR
VAR
	iSavedMementos		: INT;
	iCurrentMemento		: INT;
	astMementos			: ARRAY [0..MAX_MEMENTOS] OF ST_DocumentMemento;
END_VAR

VAR CONSTANT
	MAX_MEMENTOS		: INT := 100;
END_VAR

METHOD addMemento : BOOL
VAR_INPUT
	in_stMemento		: ST_DocumentMemento;
END_VAR

VAR
	iIndexToStore		: INT;
	i					: INT;
END_VAR
iIndexToStore := iCurrentMemento + 1;

IF iIndexToStore > MAX_MEMENTOS THEN
	
	RETURN;
	
END_IF

astMementos[iIndexToStore] := in_stMemento;

iCurrentMemento := iIndexToStore;
iSavedMementos 	:= iIndexToStore;

FOR i:= iIndexToStore + 1 TO  MAX_MEMENTOS DO
	MEMSET(destAddr:= ADR(astMementos[i]), fillByte:= 0, n:= SIZEOF(astMementos[i]));
END_FOR
END_METHOD

METHOD redoMemento : REFERENCE TO ST_DocumentMemento;
VAR_INPUT
END_VAR
IF iCurrentMemento >= iSavedMementos THEN
	
	ADSLOGSTR(msgCtrlMask:= ADSLOG_MSGTYPE_ERROR, msgFmtStr:= 'Redo not possible.', strArg:= '');
	RETURN;
	
END_IF

iCurrentMemento := iCurrentMemento + 1;
redoMemento REF= astMementos[iCurrentMemento];
END_METHOD

METHOD undoMemento : REFERENCE TO ST_DocumentMemento;
VAR_INPUT
END_VAR
IF iCurrentMemento  <= 0 THEN
	
	ADSLOGSTR(msgCtrlMask:= ADSLOG_MSGTYPE_ERROR, msgFmtStr:= 'Undo not possible.', strArg:= '');
	RETURN;
	
END_IF

iCurrentMemento := iCurrentMemento - 1;
undoMemento REF= astMementos[iCurrentMemento];
END_METHOD

END_FUNCTION_BLOCK

// ---- Observer/PRG_SampleObserver.TcPOU
PROGRAM PRG_SampleObserver
VAR
	fbPublisher					: FB_Publisher;
	fbSubscriber1				: FB_Subscriber(sName := 'anton');
	fbSubscriber2				: FB_Subscriber(sName := 'beton');
	
	bSubscribe1					: BOOL;
	bUnsubscribe1				: BOOL;
	bSubscribe2					: BOOL;
	bUnsubscribe2				: BOOL;
	
	bNotify				: BOOL;
END_VAR

IF bSubscribe1 THEN
	
	bSubscribe1 := FALSE;
	fbPublisher.subscribe(fbSubscriber1);
	
END_IF

IF bUnsubscribe1 THEN
	
	bUnsubscribe1 := FALSE;
	fbPublisher.unsubscribe(fbSubscriber1);
	
END_IF

IF bSubscribe2 THEN
	
	bSubscribe2 := FALSE;
	fbPublisher.subscribe(fbSubscriber2);
	
END_IF

IF bUnsubscribe2 THEN
	
	bUnsubscribe2 := FALSE;
	fbPublisher.unsubscribe(fbSubscriber2);
	
END_IF

IF bNotify THEN
	
	bNotify := FALSE;
	fbPublisher.notifySubscriber();
	
END_IF

END_PROGRAM

// ---- Observer/Publisher/FB_Publisher.TcPOU
FUNCTION_BLOCK FB_Publisher
VAR_INPUT
END_VAR
VAR_OUTPUT
END_VAR
VAR
	_sContent					: STRING;
	_aipSubscribers				: ARRAY[0..MAX_SUBSCRIBERS] OF I_Subscriber;
END_VAR

VAR CONSTANT
	MAX_SUBSCRIBERS				: INT := 10;
END_VAR

METHOD notifySubscriber : BOOL
VAR_INPUT
END_VAR
VAR
	i						: INT;
END_VAR
FOR i:= 0 TO MAX_SUBSCRIBERS DO
	
	IF (_aipSubscribers[i] <> 0) THEN
		
		_aipSubscribers[i].update(in_sContent := CONCAT('New content available: ' , TO_STRING(_sContent)));
		
	END_IF

END_FOR
END_METHOD

PROPERTY sContent : STRING
GET
sContent := _sContent;
END_GET
SET
_sContent := sContent;
END_SET
END_PROPERTY

METHOD subscribe : BOOL
VAR_INPUT
	in_ipSubscriber		: I_Subscriber;
END_VAR

VAR
	i						: INT;
	iPossibleIndexToStore	: INT;
	bPossibleSubSpotFound	: BOOL;
END_VAR
subscribe				:= FALSE;
bPossibleSubSpotFound	:= FALSE;

// Search for free subscriber space
FOR i:= 0 TO MAX_SUBSCRIBERS DO
	
	// Find free subscriber spot
	IF (_aipSubscribers[i] = 0) AND NOT bPossibleSubSpotFound THEN
		
		bPossibleSubSpotFound := TRUE;
		iPossibleIndexToStore := i;
		
	END_IF
	
	// Already subscribed
	IF _aipSubscribers[i] = in_ipSubscriber THEN
		
		ADSLOGSTR(msgCtrlMask:= ADSLOG_MSGTYPE_ERROR, msgFmtStr:= 'From Publisher Already subscribed!', strArg:= '');
		subscribe := TRUE;
		RETURN;
		
	END_IF

END_FOR

IF bPossibleSubSpotFound THEN

	ADSLOGSTR(msgCtrlMask:= ADSLOG_MSGTYPE_ERROR, msgFmtStr:= 'From Publisher subscribtion successfull', strArg:= '');
	_aipSubscribers[iPossibleIndexToStore] := in_ipSubscriber;
	subscribe := TRUE;
	RETURN;
ELSE
	
	ADSLOGSTR(msgCtrlMask:= ADSLOG_MSGTYPE_ERROR, msgFmtStr:= 'From Publisher all subscrictions used', strArg:= '');

END_IF
END_METHOD

METHOD unsubscribe : BOOL
VAR_INPUT
	in_ipSubscriber		: I_Subscriber;
END_VAR

VAR
	i						: INT;
END_VAR
unsubscribe				:= FALSE;

// Search for subscriber
FOR i:= 0 TO MAX_SUBSCRIBERS DO
	
	// Subscriber founde
	IF _aipSubscribers[i] = in_ipSubscriber THEN
		
		_aipSubscribers[i] := 0;
		ADSLOGSTR(msgCtrlMask:= ADSLOG_MSGTYPE_ERROR, msgFmtStr:= 'From Publisher successfull unsubscribed', strArg:= '');
		unsubscribe := TRUE;
		RETURN;
		
	END_IF

END_FOR

ADSLOGSTR(msgCtrlMask:= ADSLOG_MSGTYPE_ERROR, msgFmtStr:= 'From Publisher subscribtion not found', strArg:= '');
END_METHOD

END_FUNCTION_BLOCK

// ---- Observer/Subscriber/FB_Subscriber.TcPOU
FUNCTION_BLOCK FB_Subscriber IMPLEMENTS I_Subscriber
VAR_INPUT
END_VAR
VAR_OUTPUT
END_VAR
VAR
	_sName				: STRING;
	_sPublisherContent	: STRING;
END_VAR

//FB_Init is always available implicitly and it is used primarily for initialization.
//The return value is not evaluated. For a specific influence, you can also declare the
//methods explicitly and provide additional code there with the standard initialization
//code. You can evaluate the return value.
METHOD FB_Init: BOOL
VAR_INPUT
    bInitRetains: BOOL; // TRUE: the retain variables are initialized (reset warm / reset cold)
    bInCopyCode: BOOL;  // TRUE: the instance will be copied to the copy code afterward (online change)
	sName	: STRING;   
END_VAR
_sName := sName;
END_METHOD

METHOD update : BOOL
VAR_INPUT
	in_sContent			: STRING;
END_VAR
ADSLOGSTR(msgCtrlMask:= ADSLOG_MSGTYPE_ERROR, msgFmtStr:= 'Hey its me %s, i got noftiyed with fresh new content', strArg:= _sName);
_sPublisherContent := in_sContent;
END_METHOD

END_FUNCTION_BLOCK

// ---- StatePattern/PRG_SampleState.TcPOU
PROGRAM PRG_SampleState
VAR
	fbStateMachine			:FB_StateMachine;
	sCurrentState			:STRING;
	bBtnStart				:BOOL;
	bBtnStop				:BOOL;
	bError					:BOOL;
END_VAR

fbStateMachine(
				in_bError	:= bError, 
				in_bStart	:= bBtnStart, 
				in_bStop	:= bBtnStop, 
				out_ipState	=> );

sCurrentState := fbStateMachine.out_ipState.CurrentState;

END_PROGRAM

// ---- StatePattern/FB_StateMachine.TcPOU
FUNCTION_BLOCK FB_StateMachine
VAR_INPUT
	in_bError				: BOOL;
	in_bStart				: BOOL;
	in_bStop				: BOOL;
END_VAR
VAR_OUTPUT
	out_ipState				:I_State := fbNotReadyState;
END_VAR
VAR
	fbNotReadyState			:FB_NotReadyState(THIS);
	fbReadyState			:FB_ReadyState(THIS);
	fbProcessingState		:FB_ProcessingState(THIS);
	
	fbRTrigStart			: R_TRIG;
	fbRTrigStop				: R_TRIG;
END_VAR

fbRTrigStart(CLK:= in_bStart);
fbRTrigStop(CLK:= in_bStop);


IF in_bError THEN
	out_ipState.ErrorOccured();
ELSE
	out_ipState.ErrorGone();
END_IF

IF fbRTrigStart.Q THEN
	out_ipState.StartProcess();
END_IF

IF fbRTrigStop.Q THEN
	out_ipState.StopProcess();
END_IF

PROPERTY INTERNAL NotReadyState : I_State
GET
NotReadyState := THIS^.fbNotReadyState;
END_GET
END_PROPERTY

PROPERTY INTERNAL ProcessingState : I_State
GET
ProcessingState := THIS^.fbProcessingState;
END_GET
END_PROPERTY

PROPERTY INTERNAL ReadyState : I_State
GET
ReadyState := THIS^.fbReadyState;
END_GET
END_PROPERTY

METHOD SetState : BOOL
VAR_INPUT
	newState : I_State;
END_VAR
THIS^.out_ipState := newState;
END_METHOD

END_FUNCTION_BLOCK

// ---- StatePattern/States/FB_NotReadyState.TcPOU
FUNCTION_BLOCK FB_NotReadyState IMPLEMENTS I_State
VAR_INPUT
END_VAR
VAR_OUTPUT
END_VAR
VAR
	pfbStateMachine			:POINTER TO FB_StateMachine;
END_VAR

{warning 'Add property implementation'}
PROPERTY CurrentState : STRING
GET
CurrentState := 'Not ready';
END_GET
END_PROPERTY

METHOD ErrorGone
pfbStateMachine^.SetState(pfbStateMachine^.ReadyState);
END_METHOD

METHOD ErrorOccured
// nothin happens
END_METHOD

//FB_Init is always available implicitly and it is used primarily for initialization.
//The return value is not evaluated. For a specific influence, you can also declare the
//methods explicitly and provide additional code there with the standard initialization
//code. You can evaluate the return value.
METHOD FB_Init: BOOL
VAR_INPUT
    bInitRetains: BOOL; // TRUE: the retain variables are initialized (reset warm / reset cold)
    bInCopyCode: BOOL;  // TRUE: the instance will be copied to the copy code afterward (online change)   
	pfbStateMachine	:POINTER TO FB_StateMachine;
END_VAR
THIS^.pfbStateMachine := pfbStateMachine;
END_METHOD

METHOD StartProcess
// nothin happens
END_METHOD

METHOD StopProcess
// nothin happens
END_METHOD

END_FUNCTION_BLOCK

// ---- StatePattern/States/FB_ReadyState.TcPOU
FUNCTION_BLOCK FB_ReadyState IMPLEMENTS I_State
VAR_INPUT
END_VAR
VAR_OUTPUT
END_VAR
VAR
	pfbStateMachine			:POINTER TO FB_StateMachine;
END_VAR

{warning 'Add property implementation'}
PROPERTY CurrentState : STRING
GET
CurrentState := 'Ready';
END_GET
END_PROPERTY

{warning 'Add method implementation '}
METHOD ErrorGone
// nothin happens
END_METHOD

{warning 'Add method implementation '}
METHOD ErrorOccured
pfbStateMachine^.SetState(pfbStateMachine^.NotReadyState);
END_METHOD

//FB_Init is always available implicitly and it is used primarily for initialization.
//The return value is not evaluated. For a specific influence, you can also declare the
//methods explicitly and provide additional code there with the standard initialization
//code. You can evaluate the return value.
METHOD FB_Init: BOOL
VAR_INPUT
    bInitRetains: BOOL; // TRUE: the retain variables are initialized (reset warm / reset cold)
    bInCopyCode: BOOL;  // TRUE: the instance will be copied to the copy code afterward (online change)   
	pfbStateMachine	:POINTER TO FB_StateMachine;
END_VAR
THIS^.pfbStateMachine := pfbStateMachine;
END_METHOD

{warning 'Add method implementation '}
METHOD StartProcess
pfbStateMachine^.SetState(pfbStateMachine^.ProcessingState);
END_METHOD

{warning 'Add method implementation '}
METHOD StopProcess
// nothing happens
END_METHOD

END_FUNCTION_BLOCK

// ---- StatePattern/States/FB_ProcessingState.TcPOU
FUNCTION_BLOCK FB_ProcessingState IMPLEMENTS I_State
VAR_INPUT
END_VAR
VAR_OUTPUT
END_VAR
VAR
	pfbStateMachine			:POINTER TO FB_StateMachine;
END_VAR

{warning 'Add property implementation'}
PROPERTY CurrentState : STRING
GET
CurrentState := 'Processing ...';
END_GET
END_PROPERTY

{warning 'Add method implementation '}
METHOD ErrorGone
// nothin happens
END_METHOD

{warning 'Add method implementation '}
METHOD ErrorOccured
pfbStateMachine^.SetState(pfbStateMachine^.NotReadyState);
END_METHOD

//FB_Init is always available implicitly and it is used primarily for initialization.
//The return value is not evaluated. For a specific influence, you can also declare the
//methods explicitly and provide additional code there with the standard initialization
//code. You can evaluate the return value.
METHOD FB_Init: BOOL
VAR_INPUT
    bInitRetains: BOOL; // TRUE: the retain variables are initialized (reset warm / reset cold)
    bInCopyCode: BOOL;  // TRUE: the instance will be copied to the copy code afterward (online change)   
	pfbStateMachine	:POINTER TO FB_StateMachine;
END_VAR
THIS^.pfbStateMachine := pfbStateMachine;
END_METHOD

{warning 'Add method implementation '}
METHOD StartProcess
// nothin happens
END_METHOD

{warning 'Add method implementation '}
METHOD StopProcess
pfbStateMachine^.SetState(pfbStateMachine^.ReadyState);
END_METHOD

END_FUNCTION_BLOCK

// ---- Strategy/PRG_SampleStrategy.TcPOU
PROGRAM PRG_SampleStrategy
VAR
	fbGoByCar						: FB_StrategyTravelByCar;
	fbGoByTrain						: FB_StrategyTravelByTrain;
	fbGoByBycicle					: FB_StrategyTravelByBycicle;
	
	fbTravelTimeCalculator			: FB_TravelTimeCalculator(fbGoByCar);
	
	bCalculateTime					: BOOL;
	rDistance						: REAL := 10.0;
	iActStrategy					: INT; // 0: By Car, 1: By Train, 2: By Bycicle
	iOldStrategy					: INT;
END_VAR

IF bCalculateTime THEN
	bCalculateTime := FALSE;
	fbTravelTimeCalculator.calculateTravelTime(rDistance);
END_IF

IF iActStrategy <> iOldStrategy THEN
	iOldStrategy := iActStrategy;
	
	CASE iActStrategy OF
	0:
		fbTravelTimeCalculator.SetStrategy(fbGoByCar);
	1:
		fbTravelTimeCalculator.SetStrategy(fbGoByTrain);
	2:
		fbTravelTimeCalculator.SetStrategy(fbGoByBycicle);
	ELSE
		;
	END_CASE;
END_IF

END_PROGRAM

// ---- Strategy/Strategies/FB_StrategyTravelByCar.TcPOU
FUNCTION_BLOCK FB_StrategyTravelByCar IMPLEMENTS I_Strategy
VAR_INPUT
END_VAR
VAR_OUTPUT
END_VAR
VAR
END_VAR

METHOD execute
VAR_INPUT
	in_rDistance		:REAL;
END_VAR
ADSLOGSTR(msgCtrlMask:= ADSLOG_MSGTYPE_ERROR, msgFmtStr:= 'Travel time by car: %s min', strArg:= TO_STRING(in_rDistance * 0.7));
END_METHOD

END_FUNCTION_BLOCK

// ---- Strategy/Strategies/FB_StrategyTravelByTrain.TcPOU
FUNCTION_BLOCK FB_StrategyTravelByTrain IMPLEMENTS I_Strategy
VAR_INPUT
END_VAR
VAR_OUTPUT
END_VAR
VAR
END_VAR

METHOD execute
VAR_INPUT
	in_rDistance		:REAL;
END_VAR
ADSLOGSTR(msgCtrlMask:= ADSLOG_MSGTYPE_ERROR, msgFmtStr:= 'Travel time by train: %s min', strArg:= TO_STRING(in_rDistance * 1.5));
END_METHOD

END_FUNCTION_BLOCK

// ---- Strategy/Strategies/FB_StrategyTravelByBycicle.TcPOU
FUNCTION_BLOCK FB_StrategyTravelByBycicle IMPLEMENTS I_Strategy
VAR_INPUT
END_VAR
VAR_OUTPUT
END_VAR
VAR
END_VAR

METHOD execute
VAR_INPUT
	in_rDistance		:REAL;
END_VAR
ADSLOGSTR(msgCtrlMask:= ADSLOG_MSGTYPE_ERROR, msgFmtStr:= 'Travel time by bycicle: %s min', strArg:= TO_STRING(in_rDistance * 4.0));
END_METHOD

END_FUNCTION_BLOCK

// ---- Strategy/FB_TravelTimeCalculator.TcPOU
FUNCTION_BLOCK FB_TravelTimeCalculator
VAR_INPUT
END_VAR
VAR_OUTPUT
END_VAR
VAR
	ipStrategy				: I_Strategy;
END_VAR

METHOD calculateTravelTime : BOOL
VAR_INPUT
	in_rDistance		:REAL;
END_VAR
ipStrategy.execute(in_rDistance);
END_METHOD

//FB_Init is always available implicitly and it is used primarily for initialization.
//The return value is not evaluated. For a specific influence, you can also declare the
//methods explicitly and provide additional code there with the standard initialization
//code. You can evaluate the return value.
METHOD FB_Init: BOOL
VAR_INPUT
    bInitRetains: BOOL; // TRUE: the retain variables are initialized (reset warm / reset cold)
    bInCopyCode: BOOL;  // TRUE: the instance will be copied to the copy code afterward (online change)   
	ipStrategy	: I_Strategy;
END_VAR
THIS^.ipStrategy := ipStrategy;
END_METHOD

METHOD SetStrategy : BOOL
VAR_INPUT
	in_ipNewStrategy	: I_Strategy;
END_VAR
THIS^.ipStrategy := in_ipNewStrategy;
END_METHOD

END_FUNCTION_BLOCK

// ---- Visitor/FB_ElementA.TcPOU
FUNCTION_BLOCK FB_ElementA IMPLEMENTS I_VisitibleElement
VAR_INPUT
END_VAR
VAR_OUTPUT
END_VAR
VAR
END_VAR

METHOD accept
VAR_INPUT
	in_ipVisitor	: I_Visitor;
END_VAR
in_ipVisitor.VisitElementA(in_fbElementA:= THIS^);
END_METHOD

END_FUNCTION_BLOCK

// ---- Visitor/FB_ElementB.TcPOU
FUNCTION_BLOCK FB_ElementB IMPLEMENTS I_VisitibleElement
VAR_INPUT
END_VAR
VAR_OUTPUT
END_VAR
VAR
END_VAR

METHOD accept
VAR_INPUT
	in_ipVisitor	: I_Visitor;
END_VAR
in_ipVisitor.VisitElementB(in_fbElementB:= THIS^);
END_METHOD

END_FUNCTION_BLOCK

// ---- Visitor/FB_Visitor.TcPOU
FUNCTION_BLOCK FB_Visitor IMPLEMENTS I_Visitor
VAR_INPUT
END_VAR
VAR_OUTPUT
END_VAR
VAR
END_VAR

METHOD VisitElementA
VAR_INPUT
	in_fbElementA	: FB_ElementA;
END_VAR
ADSLOGSTR(msgCtrlMask:= ADSLOG_MSGTYPE_ERROR, msgFmtStr:= 'I visit Element A right now', strArg:= '');
END_METHOD

{warning 'Add method implementation '}
METHOD VisitElementB
VAR_INPUT
	in_fbElementB	: FB_ElementB;
END_VAR
ADSLOGSTR(msgCtrlMask:= ADSLOG_MSGTYPE_ERROR, msgFmtStr:= 'I visit Element B right now', strArg:= '');
END_METHOD

END_FUNCTION_BLOCK

// ---- Visitor/PRG_SampleVisitor.TcPOU
PROGRAM PRG_SampleVisitor
VAR
	fbExporter					: FB_Visitor;
	fbElementA					: FB_ElementA;
	fbElementB					: FB_ElementB;	

	bEnable						:BOOL;
END_VAR

//*************************************************************
// Disable Test enviroment
//*************************************************************	
	IF NOT bEnable THEN
		
		RETURN;
		
	END_IF
	
//*************************************************************
// Call Objects
//*************************************************************
	fbElementA.accept(fbExporter);
	fbElementB.accept(fbExporter);

END_PROGRAM
